// TIA Portal V16 export
// export: Created 2022-09-01T14:26:56.4935968Z, ExportSetting WithDefaults, DisplayName Totally Integrated Automation Portal, DisplayVersion V16, DisplayName TIA Portal Version Control Interface, DisplayVersion V16, DisplayName TIA Portal Openness, DisplayVersion V16, DisplayName STEP 7 Professional, DisplayVersion V16, DisplayName STEP 7 Safety, DisplayVersion V16, DisplayName WinCC Advanced, DisplayVersion V16
FUNCTION "Controlo_Ciclo_Limpeza" : Void   // FC2, LAD
{ S7_Optimized_Access := 'TRUE' }
VERSION : 0.1
// stored: AutoNumber true, IsIECCheckEnabled false, SetENOAutomatically false, UDAEnableTagReadback false
   VAR_TEMP   // added for the SCL form of the ladder/FBD networks
      _w1 : Bool;
   END_VAR
BEGIN

REGION Network 1: Hold Etapa 1
   // Devido à etapa 1 fazer reset a si mesma, foi necessário criar esta memória para indicar que tal filtro está em ciclo
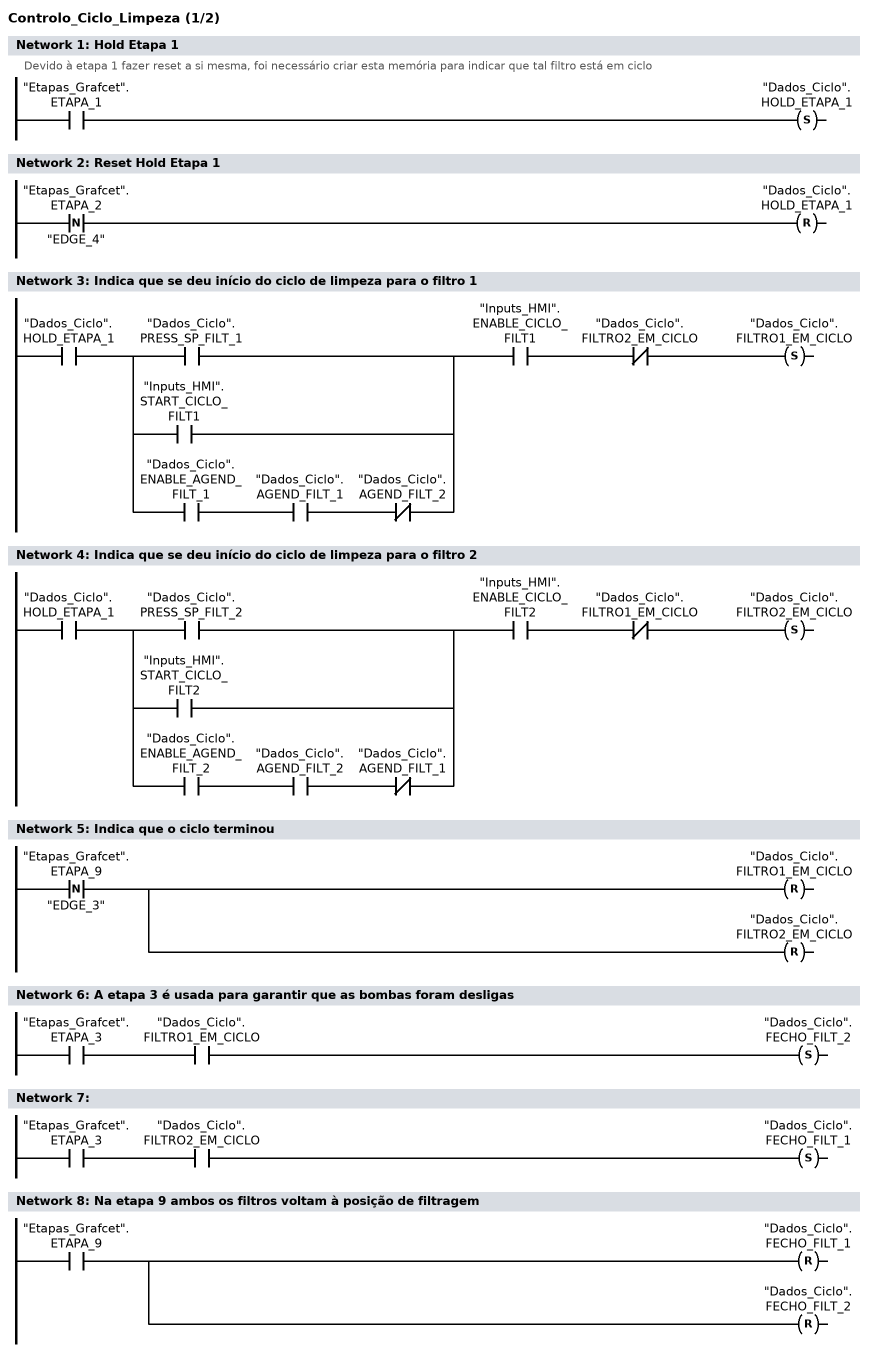
   RUNG wire#powerrail
      Contact( "Etapas_Grafcet".ETAPA_1 )
      S_Coil( "Dados_Ciclo".HOLD_ETAPA_1 )
   END_RUNG
   // the same network as SCL:
   IF "Etapas_Grafcet".ETAPA_1 THEN "Dados_Ciclo".HOLD_ETAPA_1 := TRUE; END_IF;
END_REGION

REGION Network 2: Reset Hold Etapa 1
   RUNG wire#powerrail
      N_Contact(operand := "Etapas_Grafcet".ETAPA_2, bit := "EDGE_4")
      R_Coil( "Dados_Ciclo".HOLD_ETAPA_1 )
   END_RUNG
   // the same network as SCL:
   #_w1 := NOT "Etapas_Grafcet".ETAPA_2 AND "EDGE_4";   // falling edge of "Etapas_Grafcet".ETAPA_2
   "EDGE_4" := "Etapas_Grafcet".ETAPA_2;
   IF #_w1 THEN "Dados_Ciclo".HOLD_ETAPA_1 := FALSE; END_IF;
END_REGION

REGION Network 3: Indica que se deu início do ciclo de limpeza para o filtro 1
   RUNG wire#powerrail
      Contact( "Dados_Ciclo".HOLD_ETAPA_1 )
      wire#w1
      Contact( "Dados_Ciclo".PRESS_SP_FILT_1 )
      wire#w2
      Contact( "Inputs_HMI".ENABLE_CICLO_FILT1 )
      I_Contact( "Dados_Ciclo".FILTRO2_EM_CICLO )
      S_Coil( "Dados_Ciclo".FILTRO1_EM_CICLO )
   END_RUNG
   RUNG wire#w1
      Contact( "Inputs_HMI".START_CICLO_FILT1 )
   END_RUNG wire#w2
   RUNG wire#w1
      Contact( "Dados_Ciclo".ENABLE_AGEND_FILT_1 )
      Contact( "Dados_Ciclo".AGEND_FILT_1 )
      I_Contact( "Dados_Ciclo".AGEND_FILT_2 )
   END_RUNG wire#w2
   // the same network as SCL:
   IF "Dados_Ciclo".HOLD_ETAPA_1 AND ("Dados_Ciclo".PRESS_SP_FILT_1 OR "Inputs_HMI".START_CICLO_FILT1 OR ("Dados_Ciclo".ENABLE_AGEND_FILT_1 AND "Dados_Ciclo".AGEND_FILT_1 AND NOT "Dados_Ciclo".AGEND_FILT_2)) AND "Inputs_HMI".ENABLE_CICLO_FILT1 AND NOT "Dados_Ciclo".FILTRO2_EM_CICLO THEN
       "Dados_Ciclo".FILTRO1_EM_CICLO := TRUE;
   END_IF;
END_REGION

REGION Network 4: Indica que se deu início do ciclo de limpeza para o filtro 2
   RUNG wire#powerrail
      Contact( "Dados_Ciclo".HOLD_ETAPA_1 )
      wire#w1
      Contact( "Dados_Ciclo".PRESS_SP_FILT_2 )
      wire#w2
      Contact( "Inputs_HMI".ENABLE_CICLO_FILT2 )
      I_Contact( "Dados_Ciclo".FILTRO1_EM_CICLO )
      S_Coil( "Dados_Ciclo".FILTRO2_EM_CICLO )
   END_RUNG
   RUNG wire#w1
      Contact( "Inputs_HMI".START_CICLO_FILT2 )
   END_RUNG wire#w2
   RUNG wire#w1
      Contact( "Dados_Ciclo".ENABLE_AGEND_FILT_2 )
      Contact( "Dados_Ciclo".AGEND_FILT_2 )
      I_Contact( "Dados_Ciclo".AGEND_FILT_1 )
   END_RUNG wire#w2
   // the same network as SCL:
   IF "Dados_Ciclo".HOLD_ETAPA_1 AND ("Dados_Ciclo".PRESS_SP_FILT_2 OR "Inputs_HMI".START_CICLO_FILT2 OR ("Dados_Ciclo".ENABLE_AGEND_FILT_2 AND "Dados_Ciclo".AGEND_FILT_2 AND NOT "Dados_Ciclo".AGEND_FILT_1)) AND "Inputs_HMI".ENABLE_CICLO_FILT2 AND NOT "Dados_Ciclo".FILTRO1_EM_CICLO THEN
       "Dados_Ciclo".FILTRO2_EM_CICLO := TRUE;
   END_IF;
END_REGION

REGION Network 5: Indica que o ciclo terminou
   RUNG wire#powerrail
      N_Contact(operand := "Etapas_Grafcet".ETAPA_9, bit := "EDGE_3")
      wire#w1
      R_Coil( "Dados_Ciclo".FILTRO1_EM_CICLO )
   END_RUNG
   RUNG wire#w1
      R_Coil( "Dados_Ciclo".FILTRO2_EM_CICLO )
   END_RUNG
   // the same network as SCL:
   #_w1 := NOT "Etapas_Grafcet".ETAPA_9 AND "EDGE_3";   // falling edge of "Etapas_Grafcet".ETAPA_9
   "EDGE_3" := "Etapas_Grafcet".ETAPA_9;
   IF #_w1 THEN
       "Dados_Ciclo".FILTRO1_EM_CICLO := FALSE;
       "Dados_Ciclo".FILTRO2_EM_CICLO := FALSE;
   END_IF;
END_REGION

REGION Network 6: A etapa 3 é usada para garantir que as bombas foram desligas
   RUNG wire#powerrail
      Contact( "Etapas_Grafcet".ETAPA_3 )
      Contact( "Dados_Ciclo".FILTRO1_EM_CICLO )
      S_Coil( "Dados_Ciclo".FECHO_FILT_2 )
   END_RUNG
   // the same network as SCL:
   IF "Etapas_Grafcet".ETAPA_3 AND "Dados_Ciclo".FILTRO1_EM_CICLO THEN
       "Dados_Ciclo".FECHO_FILT_2 := TRUE;
   END_IF;
END_REGION

REGION Network 7
   RUNG wire#powerrail
      Contact( "Etapas_Grafcet".ETAPA_3 )
      Contact( "Dados_Ciclo".FILTRO2_EM_CICLO )
      S_Coil( "Dados_Ciclo".FECHO_FILT_1 )
   END_RUNG
   // the same network as SCL:
   IF "Etapas_Grafcet".ETAPA_3 AND "Dados_Ciclo".FILTRO2_EM_CICLO THEN
       "Dados_Ciclo".FECHO_FILT_1 := TRUE;
   END_IF;
END_REGION

REGION Network 8: Na etapa 9 ambos os filtros voltam à posição de filtragem
   RUNG wire#powerrail
      Contact( "Etapas_Grafcet".ETAPA_9 )
      wire#w1
      R_Coil( "Dados_Ciclo".FECHO_FILT_1 )
   END_RUNG
   RUNG wire#w1
      R_Coil( "Dados_Ciclo".FECHO_FILT_2 )
   END_RUNG
   // the same network as SCL:
   IF "Etapas_Grafcet".ETAPA_9 THEN
       "Dados_Ciclo".FECHO_FILT_1 := FALSE;
       "Dados_Ciclo".FECHO_FILT_2 := FALSE;
   END_IF;
END_REGION

REGION Network 9: Set à paragem de ciclo
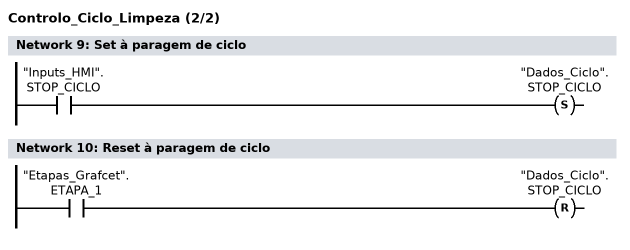
   RUNG wire#powerrail
      Contact( "Inputs_HMI".STOP_CICLO )
      S_Coil( "Dados_Ciclo".STOP_CICLO )
   END_RUNG
   // the same network as SCL:
   IF "Inputs_HMI".STOP_CICLO THEN "Dados_Ciclo".STOP_CICLO := TRUE; END_IF;
END_REGION

REGION Network 10: Reset à paragem de ciclo
   RUNG wire#powerrail
      Contact( "Etapas_Grafcet".ETAPA_1 )
      R_Coil( "Dados_Ciclo".STOP_CICLO )
   END_RUNG
   // the same network as SCL:
   IF "Etapas_Grafcet".ETAPA_1 THEN "Dados_Ciclo".STOP_CICLO := FALSE; END_IF;
END_REGION
END_FUNCTION
